(* Logix 5000 project; controller Drives_Line1 1756-L72 rev 20.13; software revision 20.04; part 15 of 21 *)
(* tags used below, declared in another part *)
   Bridle_03_Rev_mm : REAL;
   Bridle_03_SpdTrimMPS : REAL;
   Bridle_03_SpdTrimPct : REAL;
   Bridle_03a_FBCounts_mm : REAL;
   Bridle_03a_RPMPerMPS : REAL;
   Bridle_03b_RPMPerMPS : REAL;
   PulsReset_PID : TIMER;
   TimeOn_PIDOn : TIMER;
   zBridle_03_EncRes : DINT;
   zBridle_03_Ki_SpdTrim : REAL;
   zBridle_03_Kp_SpdTrim : REAL;
   zBridle_03_Kp_Treg : REAL;
   zBridle_03_MaxAccDec : REAL;
   zBridle_03_MaxTrimSpdTrim : REAL;
   zBridle_03_MinTrimSpdTrim : REAL;
   zBridle_03_Trim_HL : REAL;
   zBridle_03_Trim_LL : REAL;
   zBridle_03_WLD_Treg : REAL;
   Bridle_03 : UDT_Bridle_2M;
   LineConfig : UDT_Config_Line;
   LineCtrl : UDT_Control_Line;
   Out_Feedbacks : UDT_Fdbks;
   Out_Status : UDT_Status;
   TestConfig_Bridle_03a : UDT_Config_Bridle;
   TestConfig_Bridle_03b : UDT_Config_Bridle;
   TM2 : UDT_TM;
   zConfigFromMaster : BOOL;
   zPi : REAL;
(* P17_Bridle_03, continued *)

ROUTINE R05_Control   (* ladder *)
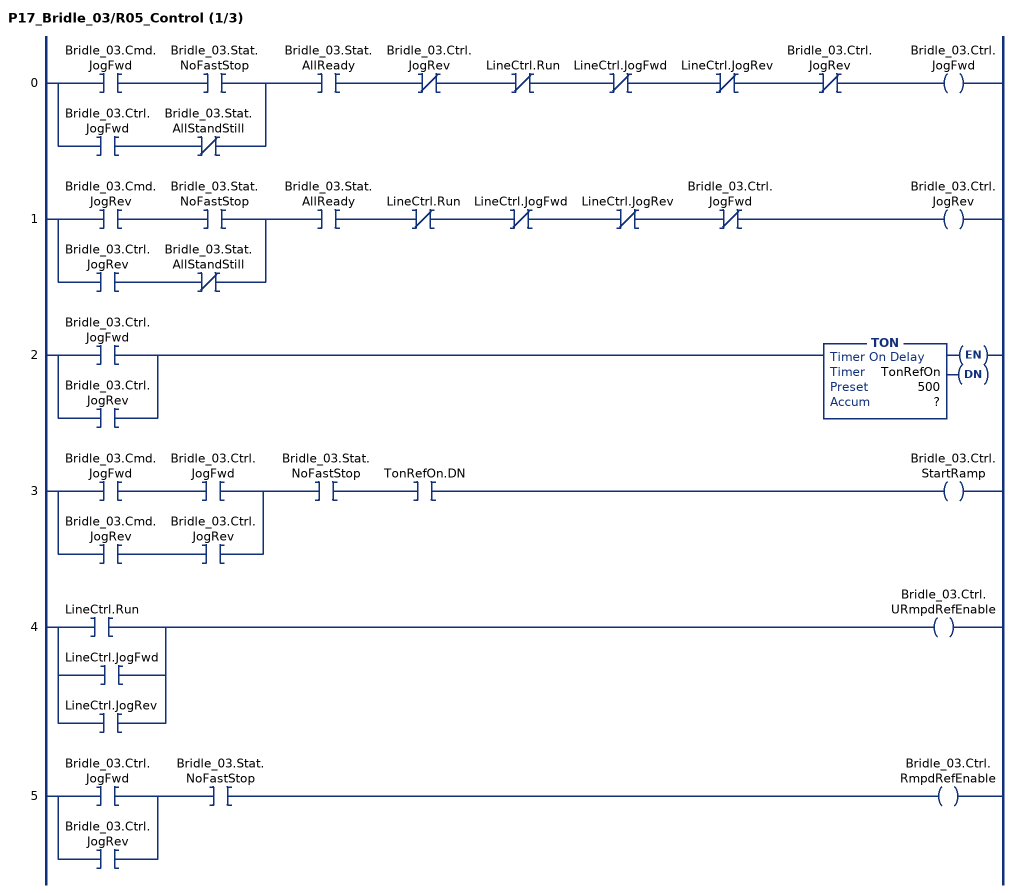
   0: [XIC(Bridle_03.Cmd.JogFwd) XIC(Bridle_03.Stat.NoFastStop) ,XIC(Bridle_03.Ctrl.JogFwd) XIO(Bridle_03.Stat.AllStandStill) ]XIC(Bridle_03.Stat.AllReady)XIO(Bridle_03.Ctrl.JogRev)XIO(LineCtrl.Run)XIO(LineCtrl.JogFwd)XIO(LineCtrl.JogRev)XIO(Bridle_03.Ctrl.JogRev)OTE(Bridle_03.Ctrl.JogFwd);
   1: [XIC(Bridle_03.Cmd.JogRev) XIC(Bridle_03.Stat.NoFastStop) ,XIC(Bridle_03.Ctrl.JogRev) XIO(Bridle_03.Stat.AllStandStill) ]XIC(Bridle_03.Stat.AllReady)XIO(LineCtrl.Run)XIO(LineCtrl.JogFwd)XIO(LineCtrl.JogRev)XIO(Bridle_03.Ctrl.JogFwd)OTE(Bridle_03.Ctrl.JogRev);
   2: [XIC(Bridle_03.Ctrl.JogFwd) ,XIC(Bridle_03.Ctrl.JogRev) ]TON(TonRefOn,?,?);
   3: [XIC(Bridle_03.Cmd.JogFwd) XIC(Bridle_03.Ctrl.JogFwd) ,XIC(Bridle_03.Cmd.JogRev) XIC(Bridle_03.Ctrl.JogRev) ]XIC(Bridle_03.Stat.NoFastStop)XIC(TonRefOn.DN)OTE(Bridle_03.Ctrl.StartRamp);
   4: [XIC(LineCtrl.Run) ,XIC(LineCtrl.JogFwd) ,XIC(LineCtrl.JogRev) ]OTE(Bridle_03.Ctrl.URmpdRefEnable);
   5: [XIC(Bridle_03.Ctrl.JogFwd) ,XIC(Bridle_03.Ctrl.JogRev) ]XIC(Bridle_03.Stat.NoFastStop)OTE(Bridle_03.Ctrl.RmpdRefEnable);
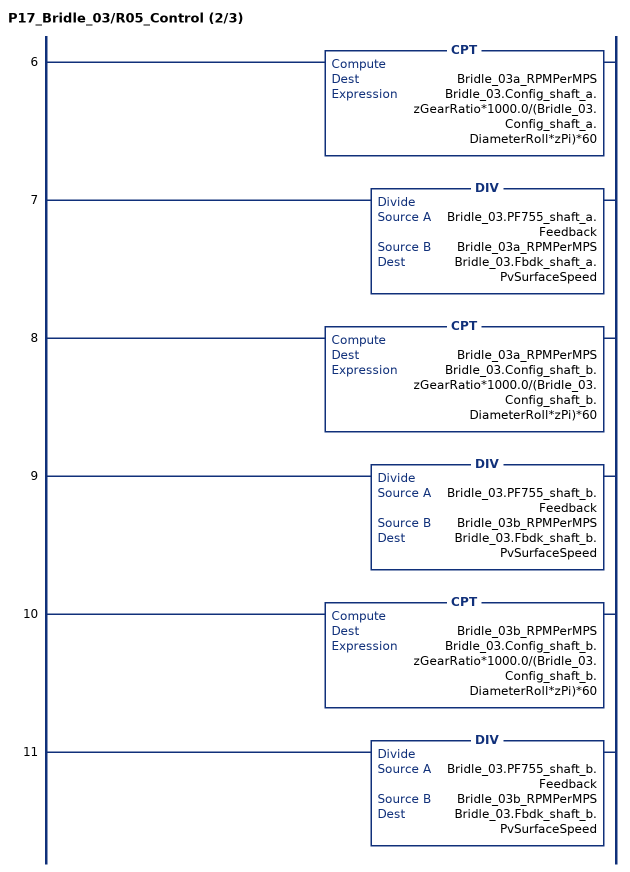
   6: CPT(Bridle_03a_RPMPerMPS,Bridle_03.Config_shaft_a.zGearRatio*1000.0/(Bridle_03.Config_shaft_a.DiameterRoll*zPi)*60);
   7: DIV(Bridle_03.PF755_shaft_a.Feedback,Bridle_03a_RPMPerMPS,Bridle_03.Fbdk_shaft_a.PvSurfaceSpeed);
   8: CPT(Bridle_03a_RPMPerMPS,Bridle_03.Config_shaft_b.zGearRatio*1000.0/(Bridle_03.Config_shaft_b.DiameterRoll*zPi)*60);
   9: DIV(Bridle_03.PF755_shaft_b.Feedback,Bridle_03b_RPMPerMPS,Bridle_03.Fbdk_shaft_b.PvSurfaceSpeed);
   10: CPT(Bridle_03b_RPMPerMPS,Bridle_03.Config_shaft_b.zGearRatio*1000.0/(Bridle_03.Config_shaft_b.DiameterRoll*zPi)*60);
   11: DIV(Bridle_03.PF755_shaft_b.Feedback,Bridle_03b_RPMPerMPS,Bridle_03.Fbdk_shaft_b.PvSurfaceSpeed);
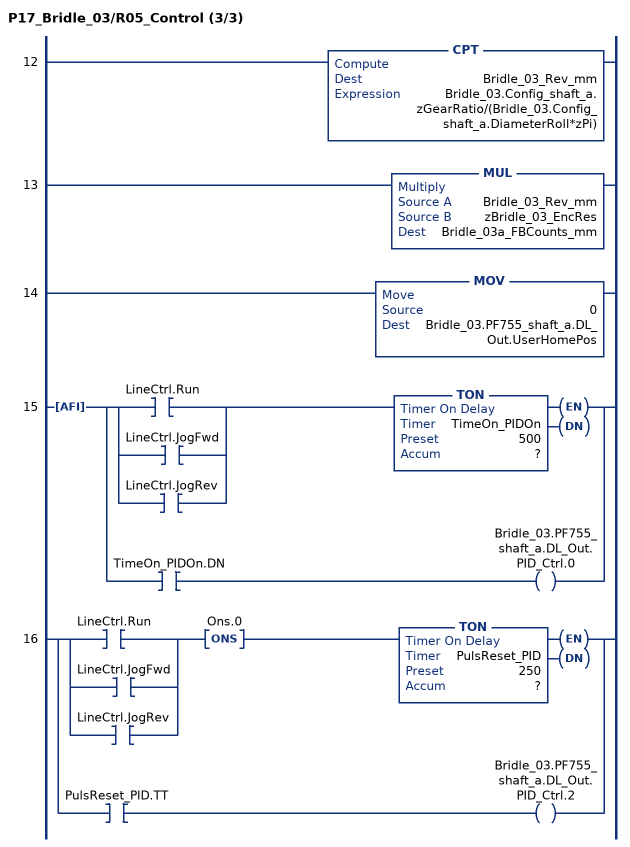
   12: CPT(Bridle_03_Rev_mm,Bridle_03.Config_shaft_a.zGearRatio/(Bridle_03.Config_shaft_a.DiameterRoll*zPi));
   13: MUL(Bridle_03_Rev_mm,zBridle_03_EncRes,Bridle_03a_FBCounts_mm);
   14: MOV(0,Bridle_03.PF755_shaft_a.DL_Out.UserHomePos);
   15: AFI()[[XIC(LineCtrl.Run) ,XIC(LineCtrl.JogFwd) ,XIC(LineCtrl.JogRev) ] TON(TimeOn_PIDOn,?,?) ,XIC(TimeOn_PIDOn.DN) OTE(Bridle_03.PF755_shaft_a.DL_Out.PID_Ctrl.0) ];
   16: [[XIC(LineCtrl.Run) ,XIC(LineCtrl.JogFwd) ,XIC(LineCtrl.JogRev) ] ONS(Ons.0) TON(PulsReset_PID,?,?) ,XIC(PulsReset_PID.TT) OTE(Bridle_03.PF755_shaft_a.DL_Out.PID_Ctrl.2) ];
END_ROUTINE

ROUTINE R10_TenReg   (* function block diagram *)
   SHEET 1   // Scale setpoint
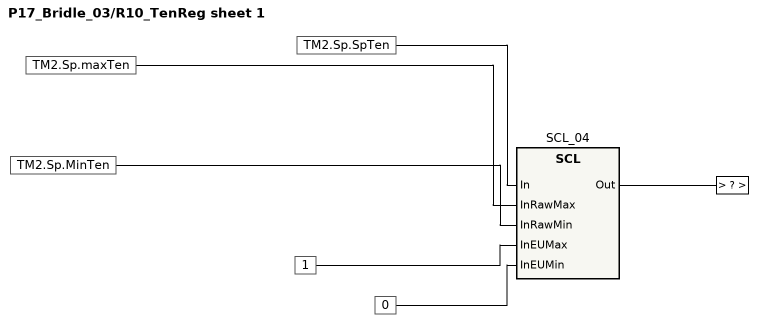
   SCL_04 : SCL(In := TM2.Sp.SpTen, InRawMax := TM2.Sp.maxTen, InRawMin := TM2.Sp.MinTen, InEUMax := 1, InEUMin := 0);
   WIRE(?) := SCL_04.Out;
   SHEET 2   // Scale tension feedback
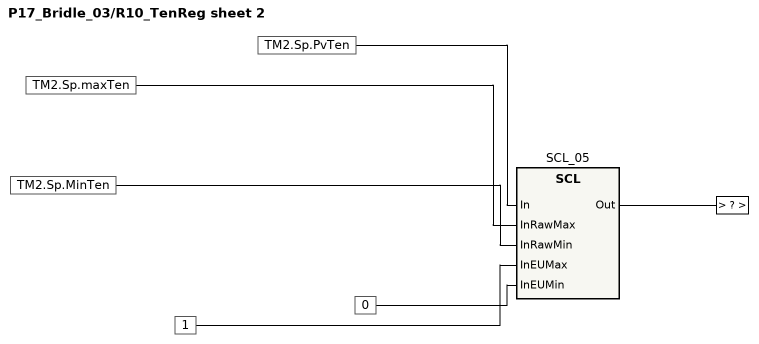
   SCL_05 : SCL(In := TM2.Sp.PvTen, InRawMax := TM2.Sp.maxTen, InRawMin := TM2.Sp.MinTen, InEUMax := 1, InEUMin := 0);
   WIRE(?) := SCL_05.Out;
   SHEET 3   // Trim limits
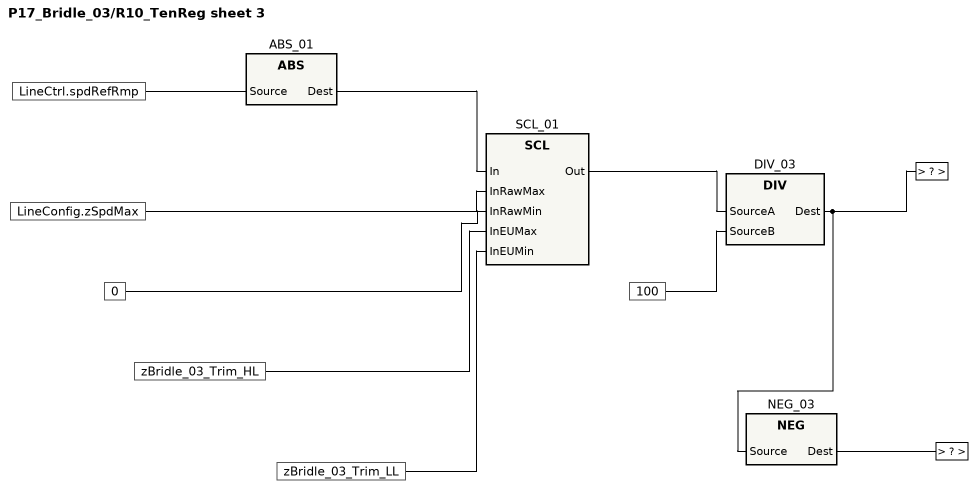
   ABS_01 : ABS(Source := LineCtrl.spdRefRmp);
   SCL_01 : SCL(In := ABS_01.Dest, InRawMax := LineConfig.zSpdMax, InRawMin := 0, InEUMax := zBridle_03_Trim_HL, InEUMin := zBridle_03_Trim_LL);
   DIV_03 : DIV(SourceA := SCL_01.Out, SourceB := 100);
   NEG_03 : NEG(Source := DIV_03.Dest);
   WIRE(?) := DIV_03.Dest;
   WIRE(?) := NEG_03.Dest;
   SHEET 4   // Tension regulator
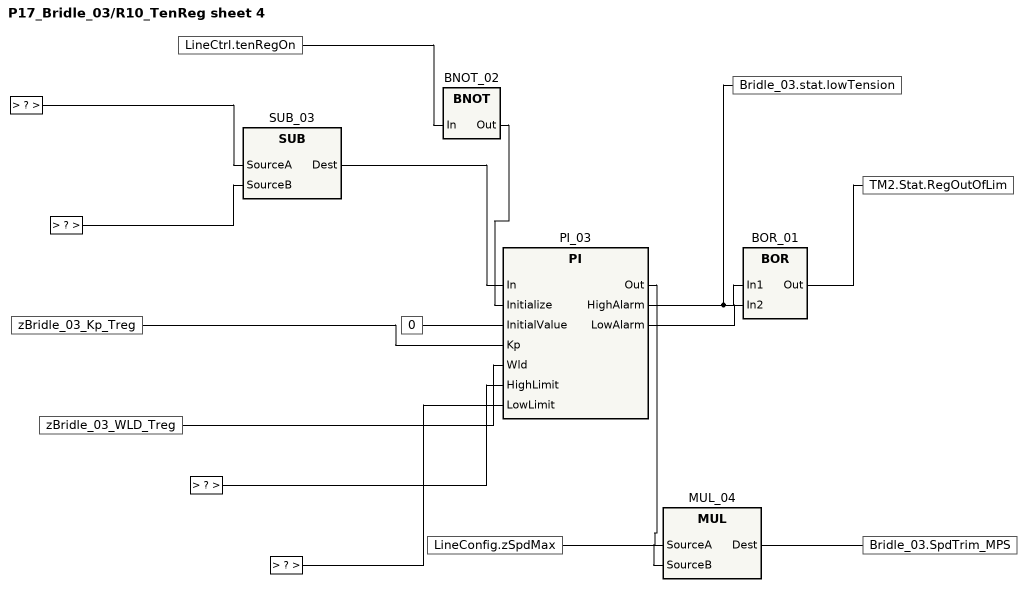
   SUB_03 : SUB(SourceA := WIRE(?), SourceB := WIRE(?));
   BNOT_02 : BNOT(In := LineCtrl.tenRegOn);
   PI_03 : PI(In := SUB_03.Dest, Initialize := BNOT_02.Out, InitialValue := 0, Kp := zBridle_03_Kp_Treg, Wld := zBridle_03_WLD_Treg, HighLimit := WIRE(?), LowLimit := WIRE(?));
   MUL_04 : MUL(SourceA := PI_03.Out, SourceB := LineConfig.zSpdMax);
   Bridle_03.stat.lowTension := PI_03.HighAlarm;
   BOR_01 : BOR(In1 := PI_03.HighAlarm, In2 := PI_03.LowAlarm);
   TM2.Stat.RegOutOfLim := BOR_01.Out;
   Bridle_03.SpdTrim_MPS := MUL_04.Dest;
END_ROUTINE

ROUTINE R11_LoadSharing   (* function block diagram *)
   SHEET 1   // Load sharing speed trim percentage
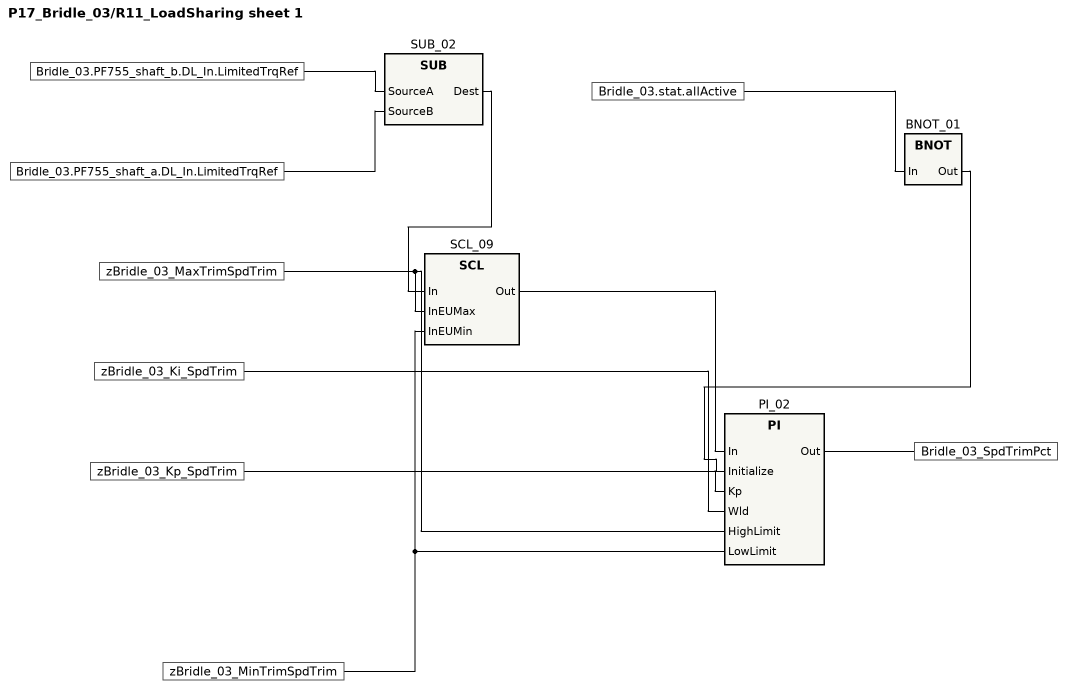
   SUB_02 : SUB(SourceA := Bridle_03.PF755_shaft_b.DL_In.LimitedTrqRef, SourceB := Bridle_03.PF755_shaft_a.DL_In.LimitedTrqRef);
   SCL_09 : SCL(In := SUB_02.Dest, InEUMax := zBridle_03_MaxTrimSpdTrim, InEUMin := zBridle_03_MinTrimSpdTrim);
   BNOT_01 : BNOT(In := Bridle_03.stat.allActive);
   PI_02 : PI(In := SCL_09.Out, Initialize := BNOT_01.Out, Kp := zBridle_03_Kp_SpdTrim, Wld := zBridle_03_Ki_SpdTrim, HighLimit := zBridle_03_MaxTrimSpdTrim, LowLimit := zBridle_03_MinTrimSpdTrim);
   Bridle_03_SpdTrimPct := PI_02.Out;
   SHEET 2   // Calculate speed trim mps
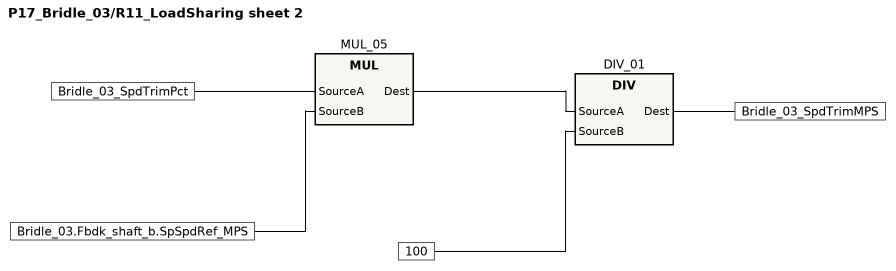
   MUL_05 : MUL(SourceA := Bridle_03_SpdTrimPct, SourceB := Bridle_03.Fbdk_shaft_b.SpSpdRef_MPS);
   DIV_01 : DIV(SourceA := MUL_05.Dest, SourceB := 100);
   Bridle_03_SpdTrimMPS := DIV_01.Dest;
END_ROUTINE

ROUTINE R12_DriveRef   (* function block diagram *)
   SHEET 1   // Select jog speed reference
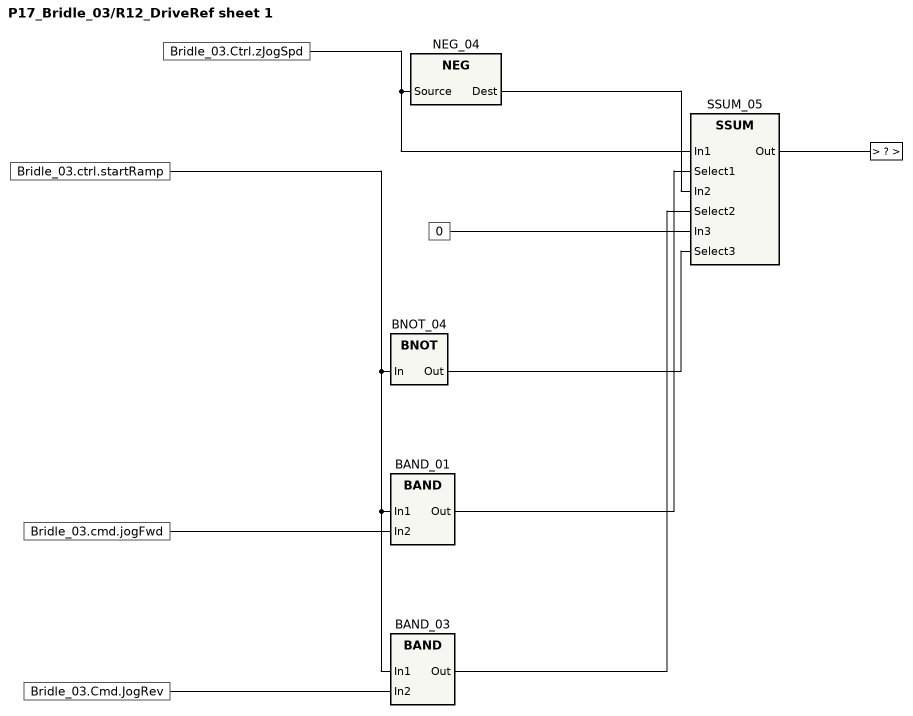
   BNOT_04 : BNOT(In := Bridle_03.ctrl.startRamp);
   BAND_01 : BAND(In1 := Bridle_03.ctrl.startRamp, In2 := Bridle_03.cmd.jogFwd);
   BAND_03 : BAND(In1 := Bridle_03.ctrl.startRamp, In2 := Bridle_03.Cmd.JogRev);
   NEG_04 : NEG(Source := Bridle_03.Ctrl.zJogSpd);
   SSUM_05 : SSUM(In1 := Bridle_03.Ctrl.zJogSpd, Select1 := BAND_01.Out, In2 := NEG_04.Dest, Select2 := BAND_03.Out, In3 := 0, Select3 := BNOT_04.Out);
   WIRE(?) := SSUM_05.Out;
   SHEET 2   // S-Curve
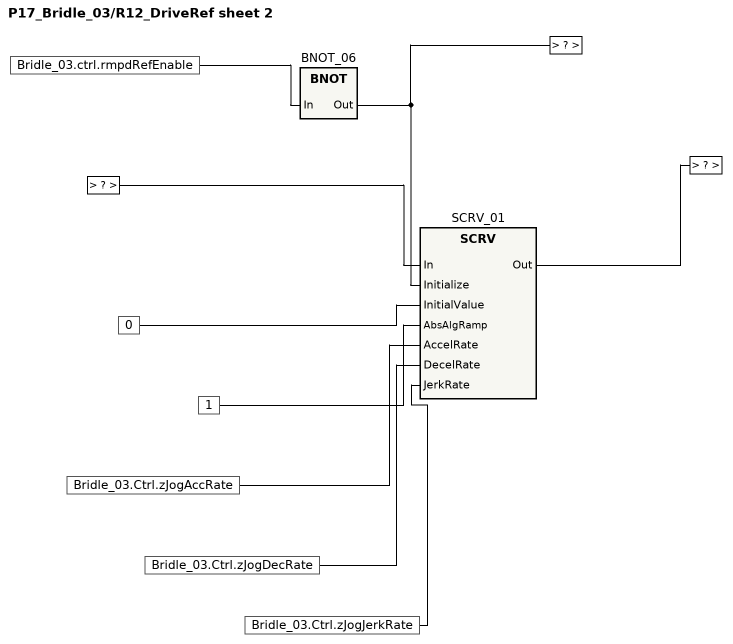
   BNOT_06 : BNOT(In := Bridle_03.ctrl.rmpdRefEnable);
   WIRE(?) := BNOT_06.Out;
   SCRV_01 : SCRV(In := WIRE(?), Initialize := BNOT_06.Out, InitialValue := 0, AbsAlgRamp := 1, AccelRate := Bridle_03.Ctrl.zJogAccRate, DecelRate := Bridle_03.Ctrl.zJogDecRate, JerkRate := Bridle_03.Ctrl.zJogJerkRate);
   WIRE(?) := SCRV_01.Out;
   SHEET 3   // Select ramped/unramped reference
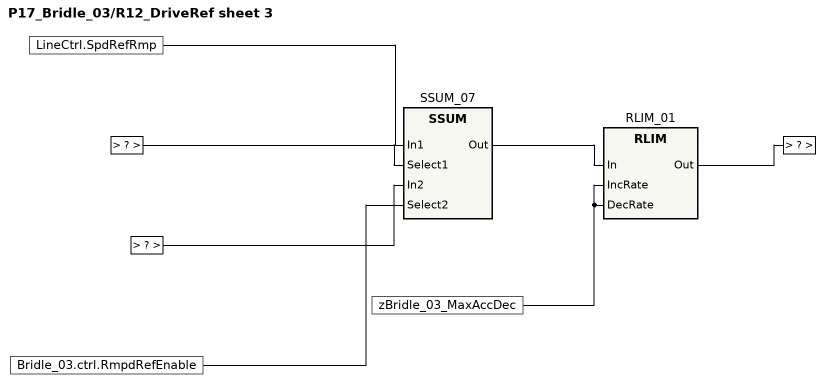
   SSUM_07 : SSUM(In1 := LineCtrl.SpdRefRmp, Select1 := WIRE(?), In2 := WIRE(?), Select2 := Bridle_03.ctrl.RmpdRefEnable);
   RLIM_01 : RLIM(In := SSUM_07.Out, IncRate := zBridle_03_MaxAccDec, DecRate := zBridle_03_MaxAccDec);
   WIRE(?) := RLIM_01.Out;
   SHEET 4   // Summarize speed reference
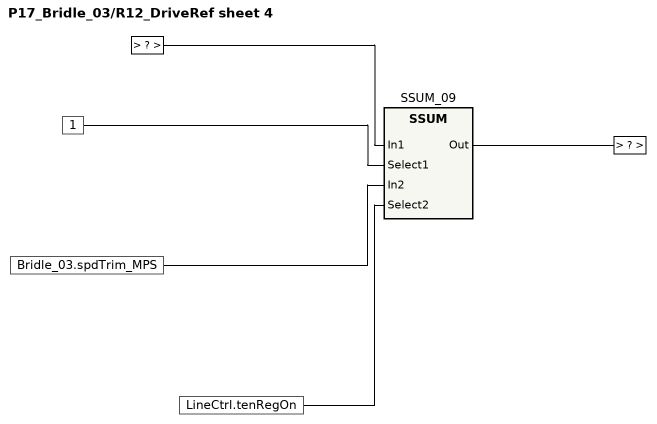
   SSUM_09 : SSUM(In1 := WIRE(?), Select1 := 1, In2 := Bridle_03.spdTrim_MPS, Select2 := LineCtrl.tenRegOn);
   WIRE(?) := SSUM_09.Out;
   SHEET 5   // Final speed reference
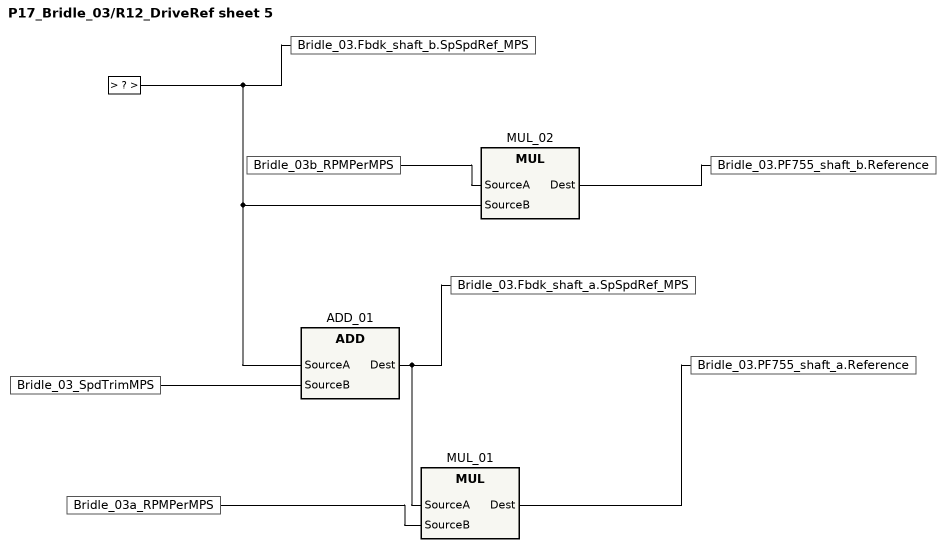
   Bridle_03.Fbdk_shaft_b.SpSpdRef_MPS := WIRE(?);
   ADD_01 : ADD(SourceA := WIRE(?), SourceB := Bridle_03_SpdTrimMPS);
   MUL_01 : MUL(SourceA := ADD_01.Dest, SourceB := Bridle_03a_RPMPerMPS);
   Bridle_03.Fbdk_shaft_a.SpSpdRef_MPS := ADD_01.Dest;
   MUL_02 : MUL(SourceA := Bridle_03b_RPMPerMPS, SourceB := WIRE(?));
   Bridle_03.PF755_shaft_a.Reference := MUL_01.Dest;
   Bridle_03.PF755_shaft_b.Reference := MUL_02.Dest;
END_ROUTINE

ROUTINE R98_ToDrive   (* ladder *)
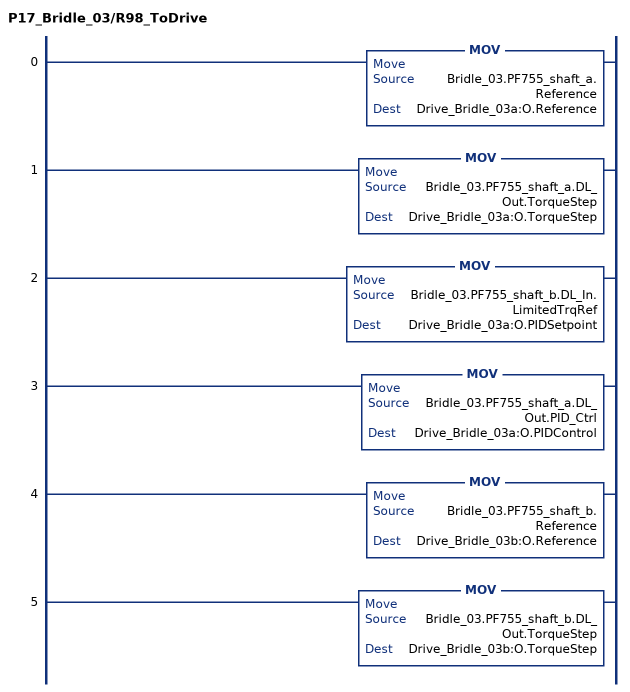
   0: MOV(Bridle_03.PF755_shaft_a.Reference,Drive_Bridle_03a:O.Reference);
   1: MOV(Bridle_03.PF755_shaft_a.DL_Out.TorqueStep,Drive_Bridle_03a:O.TorqueStep);
   2: MOV(Bridle_03.PF755_shaft_b.DL_In.LimitedTrqRef,Drive_Bridle_03a:O.PIDSetpoint);
   3: MOV(Bridle_03.PF755_shaft_a.DL_Out.PID_Ctrl,Drive_Bridle_03a:O.PIDControl);
   4: MOV(Bridle_03.PF755_shaft_b.Reference,Drive_Bridle_03b:O.Reference);
   5: MOV(Bridle_03.PF755_shaft_b.DL_Out.TorqueStep,Drive_Bridle_03b:O.TorqueStep);
END_ROUTINE

ROUTINE R999_Test   (* ladder *)
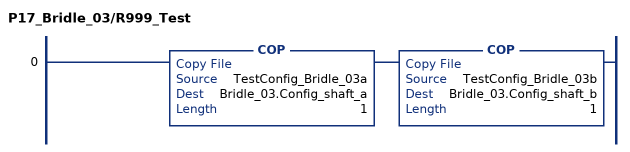
   0: COP(TestConfig_Bridle_03a,Bridle_03.Config_shaft_a,1)COP(TestConfig_Bridle_03b,Bridle_03.Config_shaft_b,1);
END_ROUTINE

ROUTINE R99_To_Master   (* ladder *)
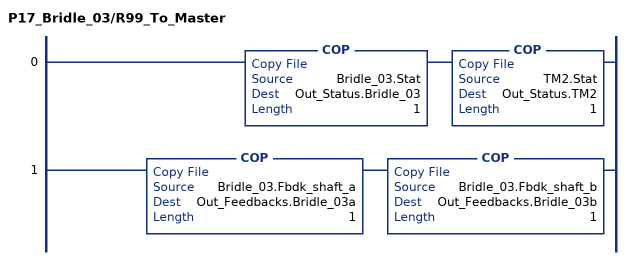
   0: COP(Bridle_03.Stat,Out_Status.Bridle_03,1)COP(TM2.Stat,Out_Status.TM2,1);
   1: COP(Bridle_03.Fbdk_shaft_a,Out_Feedbacks.Bridle_03a,1)COP(Bridle_03.Fbdk_shaft_b,Out_Feedbacks.Bridle_03b,1);
END_ROUTINE
END_PROGRAM

PROGRAM P18_Exit_Accu   (* main routine R00_Main *)
VAR
   ABS_01 : FBD_MATH_ADVANCED := (Source := 0.00068994303, Dest := 0.00068994303);
   BAND_01 : FBD_BOOLEAN_AND := (In3 := 1, In4 := 1, In5 := 1, In6 := 1, In7 := 1, In8 := 1);
   BAND_03 : FBD_BOOLEAN_AND := (In3 := 1, In4 := 1, In5 := 1, In6 := 1, In7 := 1, In8 := 1);
   BNOT_01 : FBD_BOOLEAN_NOT := (Out := 1);
   BNOT_02 : FBD_BOOLEAN_NOT := (In := 1);
   BNOT_04 : FBD_BOOLEAN_NOT := (Out := 1);
   BNOT_06 : FBD_BOOLEAN_NOT := (Out := 1);
   BOR_01 : FBD_BOOLEAN_OR;
   DIV_01 : FBD_MATH := (SourceA := 0.00068994303, SourceB := 2.0, Dest := 0.00034497152);
   DIV_02 : FBD_MATH := (SourceA := 0.5, SourceB := 2.0, Dest := 0.25);
   DIV_03 : FBD_MATH := (SourceA := 1.523458, SourceB := 100.0, Dest := 0.01523458);
   Exit_Accu_FBCounts_mm : DINT := 365;
   Exit_Accu_Rev_mm : REAL := 0.089;
   IO_State_Exit_Accu : INT := 4;
   IO_State_Tmp_Exit_Accu : INT := 16384;
   LPF_01 : FILTER_LOW_PASS := (In := 8890.0, WLag := 2.5, Order := 1, RTSTime := 1, Out := 9200.475, DeltaT := 0.05);
   MUL_01 : FBD_MATH := (SourceA := 3.9896346e-05, SourceB := 5340.0, Dest := 0.21304649);
   MUL_02 : FBD_MATH := (SourceA := 1.0, SourceB := 2.0, Dest := 2.0);
   MUL_03 : FBD_MATH := (SourceA := 29330.0, SourceB := 365.0, Dest := 10705450.0);
   MUL_04 : FBD_MATH := (SourceB := 365.0);
   MUL_05 : FBD_MATH := (SourceA := -0.00055631605, SourceB := 0.5, Dest := -0.00027815803);
   MUL_06 : FBD_MATH := (SourceA := 1000.0, SourceB := 0.089, Dest := 89.0);
   MUL_07 : FBD_MATH := (SourceA := 60.0, SourceB := 89.0, Dest := 5340.0);
   NEG_01 : FBD_MATH_ADVANCED := (Source := 0.01523458, Dest := -0.01523458);
   NEG_02 : FBD_MATH_ADVANCED := (Source := 50.0, Dest := -50.0);
   NEG_04 : FBD_MATH_ADVANCED := (Source := 0.041, Dest := -0.041);
   ons : BOOL[32];
   PI_01 : PROP_INT := (In := 9.62853, Initialize := 1, Kp := 25.0, Wld := 0.01, HighLimit := 100.0, ShapeKpPlus := 1.0, ShapeKpMinus := 1.0, ShapeWldPlus := 1.0, ShapeWldMinus := 1.0, RTSTime := 1, LowAlarm := 1, DeltaT := 0.05);
   PI_02 : PROP_INT := (In := 0.00059999526, Kp := 0.09, Wld := 0.01, HighLimit := 0.01523458, LowLimit := -0.01523458, ShapeKpPlus := 1.0, ShapeKpMinus := 1.0, ShapeWldPlus := 1.0, ShapeWldMinus := 1.0, RTSTime := 1, Out := -0.00061015034, DeltaT := 0.05);
   RLIM_01 : RATE_LIMITER := (In := 0.00034497152, IncRate := 0.5, DecRate := 0.5, RTSTime := 1, Out := 0.00034497152, DeltaT := 0.05);
   SCL_01 : SCALE := (In := 1566042.0, InRawMax := 10705450.0, InEUMax := 100.0, Out := 14.628455);
   SCL_02 : SCALE := (In := 1566047.0, InRawMax := 10705450.0, InEUMax := 29330.0, Limiting := 1, Out := 4290.5396);
   SCL_03 : SCALE := (InRawMax := 100.0, InEUMax := 0.5, Limiting := 1);
   SCL_04 : SCALE := (In := 6900.0, InRawMax := 50000.0, InEUMax := 1.0, Limiting := 1, Out := 0.138);
   SCL_05 : SCALE := (In := 6920.0, InRawMax := 50000.0, InEUMax := 1.0, Out := 0.1384);
   SCL_08 : SCALE := (In := 0.00068994303, InRawMax := 0.25, InEUMax := 10.0, InEUMin := 1.5, Limiting := 1, Out := 1.523458);
   SCRV_01 : S_CURVE := (Initialize := 1, AbsAlgRamp := 1, AccelRate := 0.08, DecelRate := 0.08, JerkRate := 0.25, RTSTime := 1, DeltaT := 0.05);
   SEL_01 : SELECT := (In1 := 50.0, In2 := 20.0, Out := 50.0);
   SSUM_03 : SELECTED_SUMMER := (In1 := 0.00034497152, Gain1 := 1.0, Select1 := 1, Gain2 := 1.0, Gain3 := 1.0, Gain4 := 1.0, Gain5 := 1.0, Gain6 := 1.0, Gain7 := 1.0, Gain8 := 1.0, Out := 0.00034497152);
   SSUM_05 : SELECTED_SUMMER := (In1 := -0.00035009556, Gain1 := 1.0, Select1 := 1, In2 := 0.00034497152, Gain2 := 1.0, Select2 := 1, Gain3 := 1.0, Gain4 := 1.0, Gain5 := 1.0, Gain6 := 1.0, Gain7 := 1.0, Gain8 := 1.0, Out := -5.1240495e-06);
   SSUM_06 : SELECTED_SUMMER := (In1 := 0.041, Gain1 := 1.0, In2 := -0.041, Gain2 := 1.0, Gain3 := 1.0, Select3 := 1, Gain4 := 1.0, Gain5 := 1.0, Gain6 := 1.0, Gain7 := 1.0, Gain8 := 1.0);
   SUB_01 : FBD_MATH := (SourceA := 14.628455, SourceB := 5.0, Dest := 9.628455);
   SUB_02 : FBD_MATH := (SourceA := 0.138, SourceB := 0.1384, Dest := -0.00040000677);
   SUB_03 : FBD_MATH := (SourceA := 0.00068994303, Dest := 0.00068994303);
   SUB_04 : FBD_MATH := (SourceA := 0.00068994303, Dest := 0.00068994303);
   TofReset : TIMER := (PRE := 1000, ACC := 1000);
   TonNoResponse : TIMER := (PRE := 2500);
   TonRefOn : TIMER := (PRE := 750);
   TonTensionOnSp : TIMER := (PRE := 1000, ACC := 1000, EN := 1, DN := 1);
   zExit_Accu_EncCounts : DINT := 4096;
   zExit_Accu_Kp_Preg : REAL := 25.0;
   zExit_Accu_Kp_Treg : REAL := 0.09;
   zExit_Accu_MaxAccDec : REAL := 0.5;
   zExit_Accu_NrOfCyl : DINT := 1;
   zExit_Accu_Pos_PreLim : REAL := 100.0;
   zExit_Accu_SpdRegMax : REAL := 50.0;
   zExit_Accu_SpdRegMin : REAL := 20.0;
   zExit_Accu_SpdTrim_HL : REAL := 10.0;
   zExit_Accu_SpdtRim_LL : REAL := 1.5;
   zExit_Accu_WLD_Preg : REAL := 0.01;
   zExit_Accu_WLD_Treg : REAL := 0.01;
   zExit_Accu_WLD_Treg_FB : REAL := 2.5;
   zNoMaster : BOOL := 1;
   zTM3_Tens_Offset : REAL := 500.0;
END_VAR

ROUTINE R00_Main   (* ladder *)
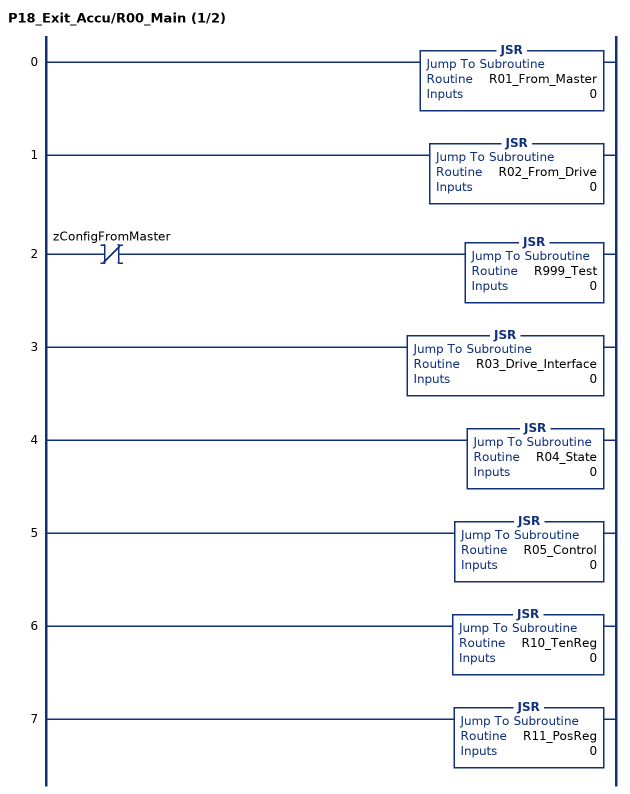
   0: JSR(R01_From_Master,0);
   1: JSR(R02_From_Drive,0);
   2: XIO(zConfigFromMaster)JSR(R999_Test,0);
   3: JSR(R03_Drive_Interface,0);
   4: JSR(R04_State,0);
   5: JSR(R05_Control,0);
   6: JSR(R10_TenReg,0);
   7: JSR(R11_PosReg,0);
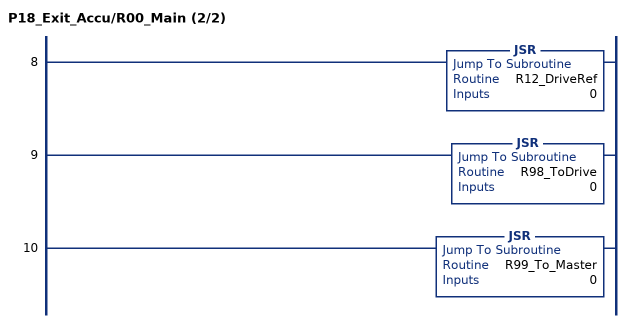
   8: JSR(R12_DriveRef,0);
   9: JSR(R98_ToDrive,0);
   10: JSR(R99_To_Master,0);
END_ROUTINE
